{attribute 'GeneratedUsingTerminal: EJ5002-0000-0017'}
{attribute addProperty BoxType "EJ5002-0000-0017"}
{attribute addProperty Id "Data_errorBOOL1Frame_errorBOOL1Power_failureBOOL1Data_mismatchBOOL1Sync_errorBOOL1TxPDO_StateBOOL1TxPDO_ToggleBOOL1"}
{attribute addProperty CRC "3225298069"}
{attribute addProperty Size "7"}
TYPE Status_C03E2495 :
STRUCT
	{attribute addProperty Name "Data_error"}
	Data_error : BOOL;
	{attribute addProperty Name "Frame_error"}
	Frame_error : BOOL;
	{attribute addProperty Name "Power_failure"}
	Power_failure : BOOL;
	{attribute addProperty Name "Data_mismatch"}
	Data_mismatch : BOOL;
	{attribute addProperty Name "Sync_error"}
	Sync_error : BOOL;
	{attribute addProperty Name "TxPDO_State"}
	TxPDO_State : BOOL;
	{attribute addProperty Name "TxPDO_Toggle"}
	TxPDO_Toggle : BOOL;
END_STRUCT
END_TYPE

(* stored: Version 1.2.0.0, ProductVersion 3.1.4024.9
   DUT Status_C03E2495: Id {8190d34b-a8f3-4530-b4e5-5583f46e5b82} *)
